FUNCTION_BLOCK EnableGroup EXTENDS TaskBase
VAR_INPUT
END_VAR
VAR_OUTPUT
END_VAR
VAR
	groupEnable			: MC_GroupEnable;
	_caGroup			: ICollisionGroup;
	_enableGroup : BOOL;
END_VAR

{analysis -2}

METHOD Abort : BOOL
groupEnable.Execute := FALSE;
Abort := TRUE;
State := 0;
END_METHOD

METHOD Cycle : HRESULT
VAR_INPUT
END_VAR
Cycle := S_OK;
CASE State OF
	0:
		IF _enableGroup THEN
			Cycle := S_PENDING;
			_Done := FALSE;
			_Error := FALSE;
			_Busy := TRUE;
			groupEnable.Execute := TRUE;
			IF groupEnable.Busy THEN
				State := 10;
				_enableGroup := FALSE;
				Logger.Send(TC_EVENTS.XtsCaGroupEvents.CAGroupEnabling,'');
			END_IF
		END_IF
	
	10:
		IF NOT groupEnable.Busy THEN
			IF groupEnable.Done THEN
				_Done := TRUE;
				Logger.Send(TC_EVENTS.XtsCaGroupEvents.CAGroupEnabled,'');
			ELSIF groupEnable.Error THEN
				_Error := TRUE;
				Logger.Send(TC_EVENTS.XtsCaGroupEvents.CAGroupEnableError,'');
			END_IF
			_Busy := FALSE;
			groupEnable.Execute := false;
			State := 0;
			Cycle := S_OK;
		END_IF
	ELSE
		Cycle := E_FAIL;
END_CASE


groupEnable(AxesGroup := _caGroup.GroupRef);
END_METHOD

METHOD Execute : BOOL
Execute := _enableGroup := true;
END_METHOD

METHOD FB_init : BOOL
VAR_INPUT
	bInitRetains : BOOL; // if TRUE, the retain variables are initialized (warm start / cold start)
	bInCopyCode : BOOL;  // if TRUE, the instance afterwards gets moved into the copy code (online change)
	MyCaGroup : ICollisionGroup;	
END_VAR
_caGroup := MyCaGroup;
END_METHOD

END_FUNCTION_BLOCK

(* stored: Version 1.1.0.1, ProductVersion 3.1.4024.12
   POU EnableGroup: Id {01c66182-3535-4445-8b1b-a8f549e6d0ab}, SpecialFunc None
   Method Abort: Id {8e535bd0-5fdc-4fa1-a309-8fd0da8ee400}
   Method Cycle: Id {53999691-fece-418c-ba0c-d2348e6bf666}
   Method Execute: Id {6b5a42b1-94d9-46bc-bf55-d1fbc24c1815}
   Method FB_init: Id {7ad275c7-67dd-42d2-bf9e-97af0354a9b5} *)
